(* CODESYS project heartbeat.2020.0113.1.project

Project tree, tasks and I/O mapping:
  Device : Changsha-Cyber-MI-linux, Changsha Cyber-MI Co., Ltd., version 3.5.10.40
    application Application
      libraries: Standard, * (System); SysFile, 3.5.9.0 (System); SysTypes2 Interfaces, * (System); SysShm, * (System); CAA Mathematics, * (CAA Technical Workgroup); SysTime, 3.5.9.0 (System); CAA Types Extern, 3.5.13.0 (CAA Technical Workgroup); TCP, 3.5.9.50 (3S - Smart Software Solutions GmbH); CAA Net Base Services, 3.5.14.0 (CAA Technical Workgroup); CAA DTUtil Extern, 3.5.12.0 (CAA Technical Workgroup); Util, * (System)
      task c_MainTask (cyclic, interval 10 ms, priority 20) calls prg_heartbeat, prg_data2file
      Enums/
        data type ERROR
        data type MQTT_STATE
        data type UDP_STATE_1
      data type UDP_STATE
      programs/
        program prg_heartbeat [ST]
      Function Blocks/
        function block FB_RETAIN [ST]: wr_all, SetDefault, chk_change, rd_all, is_default
        function block FB_MQTT_PUBLISH_CLIENT [ST]: m_fill_publish_buf, m_fill_connect_buf
        function block FB_DATA2FILE [ST]
      Functions/
        function Enable_120ohm_can0 [ST]
        function write_num_to_file [ST]
        function read_num_from_file [ST]
        function Enable_120ohm_can1 [ST]
        function Disable_120ohm_can0 [ST]
        function Disable_120ohm_can1 [ST]
        function Set_piv01 [ST]
        function Set_piv23 [ST]
        function set_ip [ST]
        function set_wifi_passwd [ST]
        function read_iccid [ST]
        function read_ip [ST]
        function read_sn [ST]
        function read_wifi_passwd [ST]
        function read_work_mins [ST]
        function read_location [ST]
      heartbeat/
        function fn_cyber_layer1 [ST]
        function fn_cyber_layer2 [ST]
        function fn_cyber_heartBeat [ST]
        function fn_sn_str_to_byte [ST]
        function Iccid_to_bytes [ST]
      GlobalConstants/
        global variables Constants
      program prg_data2file [ST]
    SoftMotion General Axis Pool
  libraries: VisuSymbols, 3.5.10.0 (System)
  5ce3da45-db07-42e7-a21c-a00fff4ed8f6|C:\Users\zhou\p01.bmp
  5ce3da45-db07-42e7-a21c-a00fff4ed8f6|C:\working\p01.bmp
  5ce3da45-db07-42e7-a21c-a00fff4ed8f6|C:\working\file.bmp
  text list GlobalTextList
*)

// Device/Application/UDP_STATE
TYPE UDP_STATE :
(
	INIT := 0, 	(* first State. Connections are set up *)
	SEND,		(* Send messages *)
	READ,		(* Receive messages *)
	ERROR		(* Prepare to reset connections *)
);
END_TYPE

// Device/Application/Enums/ERROR
{attribute 'qualified_only'}
//{attribute 'conditionalshow'}
//{attribute 'conditionalshow' := 'SomeText'}
//{attribute 'hide'}
TYPE ERROR : (NO_ERROR, TIME_OUT); END_TYPE

// Device/Application/Enums/MQTT_STATE
{attribute 'qualified_only'}
{attribute 'strict'}
TYPE MQTT_STATE :
(
	INIT := 0,
	CONN_SEND,
	CONN_RECV,
	READY,
	SEND,
	RECV,
	ERROR
);
END_TYPE

// Device/Application/Enums/UDP_STATE_1
TYPE UDP_STATE_1 :
(
	INIT := 0, 	(* first State. Connections are set up *)
	SEND,		(* Send messages *)
	READ,		(* Receive messages *)
	ERROR		(* Prepare to reset connections *)
);
END_TYPE

// Device/Application/GlobalConstants/Constants
{attribute 'qualified_only'}

VAR_GLOBAL CONSTANT
	RETAIN_NUM_MAX : INT := 256; 
END_VAR

// Device/Application/programs/prg_heartbeat
PROGRAM prg_heartbeat
VAR_OUTPUT
	lock_state :INT := 0;
	unlock_state :INT := 0;
	lock_unlock_level :INT := 0;
	delay_time :INT := 0;
END_VAR

VAR
	is_inited :BOOL := FALSE;
	eSTATE			: UDP_STATE; (* 状态转换变量 *)
	
	myIP		: NBS.IP_ADDR; (* MIC7001本身的IP地址 *)
	myPort		: UINT; (* MIC7001用于通信的端口 *)
	IPSend		: NBS.IP_ADDR; (* 对方的IP地址 *)
	PortSend	: UINT; (* 对方的端口 *)

	sToSend			: STRING; (* 待发送数据 *)
	sReceived		: STRING; (* 接收数据 *)
	
	UDPPeer			: NBS.UDP_Peer; (* FB UDP Peer *)
	UDPSend			: NBS.UDP_Send; (* FB UDP Send *)
	UDPReceive		: NBS.UDP_Receive; (* FB UDP Receive *)
	Peer			: CAA.HANDLE; (* Handle to the peer connection *)

	size :CAA.SIZE;	
	Writebuffer: 			ARRAY[1..200] OF BYTE;
	Readbuffer: 			ARRAY[0..1499] OF BYTE;
	ReadbufferStr: STRING;
	atcState :INT := 0;
	
	writeUdpState :INT := 0;
	readUdpState :INT := 0;
	
	i :INT;
	count :INT := 0;
	
	rtc_fb: RTC;
	dtu_set_dt_fb: dtu.SetDateAndTime;
	
	
	server_ip:STRING := '47.107.240.29';
	server_port:UINT := 34567;
	
	is_read :BOOL := FALSE;
	read_count :INT := 0;
	readFileState :INT := 0;
	ton_fb :TON;
	iccid_read_buffer :STRING;
	position :INT := -1;
	new_date:DT;
	iStat :UINT := 0;
	lac : STRING(4) := '0000';
	ci : STRING(4) := '0000';
	lenHearBeat:UINT;
	dataHearBeat:ARRAY[0..255] OF BYTE;
	ton_hb:ton; //heartbeat timer 
	bReturn:BOOL;
	lenLayer2:UINT;
	dataLayer2:ARRAY[0..255] OF BYTE;
	lenLayer1:UINT;
	lenRecvLayer1:UINT := 1500;
	dataLayer1:ARRAY[0..255] OF BYTE;
	bSN :ARRAY[0..6] OF BYTE;
	sub_str:STRING(8);
	num :UINT;
	lenHeartBeat: UINT;
	sn: STRING;
	work_time: DINT;
	dataIndex :UINT := 0;
	cntr_lac:UINT := 0;
	cntr_iccid:UINT := 0;
	cntr_recv:UINT := 0;
	dataLayern:ARRAY[1..255] OF BYTE;
	recv_size :CAA.SIZE;
	
	/// 辅助变量 
	xSend			: BOOL;
	sTmp1			: STRING;
	xEnable			: BOOL;	
	gprs_serial :CAA.HANDLE;
END_VAR

CASE iStat OF
0:
	xEnable:= TRUE;  //用于启动最下方的第70行的UDPPeer
	// 建立连接后马上转到发送状态
	IF UDPPeer.xActive THEN 
		eSTATE:= UDP_STATE.send;
	ELSIF UDPPeer.xError THEN
		eSTATE:= UDP_STATE.ERROR;
	END_IF
	
	IPSend.sAddr := server_ip;
	iStat := 2;
	
2:
	IF NOT read_iccid(ADR(iccid_read_buffer)) THEN
		iccid_read_buffer := 'iccid_null';		
	END_IF;
	iStat := 10;
	
10: //read sn
	IF NOT read_sn(ADR(sn)) THEN 
		sn := 'sn_null';
	END_IF
	
	iStat := 15;
	
15:
	read_location(ADR(lac), ADR(ci));
	iStat := 30;
30:
	work_time := read_work_mins();
	iStat := 100;
	
100:   //定时等待
	ton_fb(IN := TRUE, PT := T#10S);
	IF (ton_fb.Q) THEN
		ton_fb(IN := FALSE, PT := T#10S);
		iStat := 200;  //发送心跳
	ELSE
		iStat := 300; //发送实时数据	
	END_IF
	
200:
	bReturn := fn_cyber_heartBeat(	  //填充第三层：心跳帧
						lac_str := lac, 
						cid_str := ci, 
						ccid_str := iccid_read_buffer, 
						mins := work_time, 
						clientCode := 6,   //hengtian 95
						machineCode := 5,  //挖掘机
						pLenOut := ADR(lenHearBeat), 
						pDataOut := ADR(dataHearBeat)
	);
	
	IF NOT bReturn THEN
		RETURN;
	END_IF;

	dataIndex := dataIndex + 1;
	bReturn := fn_cyber_layer2( //填充第二层，数据层
						dataType := 1,
						paraId := 0,
						dataIndex := dataIndex,
						ver := 1,
						res1 := 0,
						LenIn := lenHearBeat,
						pDataIn := ADR(dataHearBeat),
						pLenOut := ADR(lenLayer2),
						pDataOut := ADR(dataLayer2)
	);
				
	IF NOT bReturn THEN
		RETURN;
	END_IF;

	bSN := fn_sn_str_to_byte(sn);
	bReturn := fn_cyber_layer1(    //填充第一层，设备层
						sn := ADR(bSN),
						ver := 1,
						lenIn := lenLayer2,
						pDataIn := ADR(dataLayer2),
						pLenOut := ADR(lenLayer1),
						pDataOut := ADR(dataLayer1)
	);
	
	IF NOT bReturn THEN
		RETURN;
	ELSE
		UDPSend(xExecute := FALSE);
		iStat := 500;
	END_IF;
	
300:  //sending realtime data  here
	//UDPSend(some realtime data as need);
	iStat := 100;
	
500:
	UDPSend(xExecute := TRUE, hPeer := Peer, ipAddr := IPSend, uiPort := server_port, szSize := lenLayer1, pDAta := ADR(dataLayer1));
	IF UDPSend.xDone THEN
		UDPSend(xExecute := FALSE);
		iStat := 600; 
	END_IF
	
	IF UDPSend.xError THEN  
		UDPSend(xExecute := FALSE);
		iStat := 30; 
	END_IF
	
	
600:
	UDPReceive(xEnable := TRUE, hPeer := Peer, szSize := SIZEOF(Readbuffer), pData := ADR(Readbuffer));
	IF UDPReceive.xDone THEN  //接收到数据
	 	recv_size := UDPReceive.szCount;
		UDPReceive(xEnable := FALSE);
		iStat := 30; //read mins and lca again
		IF recv_size = 25 THEN
			lock_state := BYTE_TO_INT(Readbuffer[20]);
			unlock_state := BYTE_TO_INT(Readbuffer[21]);
			lock_unlock_level := BYTE_TO_INT(Readbuffer[22]);
			delay_time := BYTE_TO_INT(Readbuffer[23]);
		END_IF
	ELSE
		cntr_recv := cntr_recv + 1;
		IF cntr_recv > 20 THEN
			cntr_recv := 0;
			iStat := 30;
		END_IF
	END_IF
	
	IF UDPReceive.xError THEN  //接收错误
		UDPReceive(xEnable := FALSE);
		recv_size := 0;
		iStat := 30; //read mins and lca again
	END_IF
END_CASE

//保持每个周期调用，维护与对方的连接关系本地端口的接收状态
UDPPeer(xEnable:= xEnable, hPeer=> Peer);
RETURN;

END_PROGRAM

// Device/Application/Functions/read_iccid
FUNCTION read_iccid : BOOL
VAR_INPUT
	iccid: POINTER TO STRING;
END_VAR

VAR
	hFile: RTS_IEC_HANDLE;
	udiOpenError: RTS_IEC_RESULT;
	udiReadError: RTS_IEC_RESULT;
	i :INT;
	iTemp: UDINT;
	udiPos: UDINT;
	str_size: __XWORD;
	udiByteRead: LWORD;

	len_of_line: INT;
	len_of_number :INT;
	magicNumber:REAL;
	check_sum:REAL:= 0;
	temp_num:REAL;
END_VAR

read_iccid := FALSE;

//检测文件是否存在
hFile := sysfileopen(szFile := '/userapp/iccid.txt', am := sysfile.AM_READ, pResult:= ADR(udiOpenError));
IF hFile = RTS_INVALID_HANDLE	THEN  //文件不存在
	RETURN;
END_IF
//文件存在，开始读取内容
udiPos := SysFileSetPos(hFile:=hFile, ulOffset := 0);
udiByteRead := sysfile.SysFileRead(hfile := hFile,pbyBuffer := iccid, ulSize := 32, pResult := ADR(udiReadError));
IF udiByteRead < 4 THEN  //读取失败
	sysfile.SysFileClose(hFile := hFile);
	RETURN;
END_IF

sysfile.SysFileClose(hFile := hFile);
read_iccid := TRUE;

END_FUNCTION

// Device/Application/Functions/read_sn
FUNCTION read_sn : BOOL
VAR_INPUT
	sn: POINTER TO STRING;
END_VAR

VAR
	hFile: RTS_IEC_HANDLE;
	udiOpenError: RTS_IEC_RESULT;
	udiReadError: RTS_IEC_RESULT;
	i :INT;
	iTemp: UDINT;
	udiPos: UDINT;
	str_size: __XWORD;
	udiByteRead: LWORD;

	len_of_line: INT;
	len_of_number :INT;
	magicNumber:REAL;
	check_sum:REAL:= 0;
	temp_num:REAL;
END_VAR

read_sn := FALSE;

//检测文件是否存在
hFile := sysfileopen(szFile := '/userapp/sn.txt', am := sysfile.AM_READ, pResult:= ADR(udiOpenError));
IF hFile = RTS_INVALID_HANDLE	THEN  //文件不存在
	RETURN;
END_IF
//文件存在，开始读取内容
udiPos := SysFileSetPos(hFile:=hFile, ulOffset := 0);
udiByteRead := sysfile.SysFileRead(hfile := hFile,pbyBuffer := sn, ulSize := 32, pResult := ADR(udiReadError));
IF udiByteRead < 4 THEN  //读取失败
	sysfile.SysFileClose(hFile := hFile);
	RETURN;
END_IF
sysfile.SysFileClose(hFile := hFile);
read_sn := TRUE;

END_FUNCTION

// Device/Application/Functions/read_location
FUNCTION read_location : BOOL
VAR_INPUT
	lac:POINTER TO STRING;
	ci:POINTER TO STRING;
END_VAR

VAR
	hFile: RTS_IEC_HANDLE;
	udiOpenError: RTS_IEC_RESULT;
	udiReadError: RTS_IEC_RESULT;
	i :INT;
	iTemp: UDINT;
	udiPos: UDINT;
	str_size: __XWORD;
	udiByteRead: LWORD;

	len_of_line: INT;
	len_of_number :INT;
	magicNumber:REAL;
	check_sum:REAL:= 0;
	temp_num:REAL;	
END_VAR

read_location := FALSE;
lac^ := '0000';
ci^ := '0000';

//检测文件是否存在
hFile := sysfileopen(szFile := '/userapp/laccid.txt', am := sysfile.AM_READ, pResult:= ADR(udiOpenError));
IF hFile = RTS_INVALID_HANDLE	THEN  //文件不存在
	RETURN;
END_IF

//文件存在，开始读取内容
udiPos := SysFileSetPos(hFile:=hFile, ulOffset := 0);
udiByteRead := sysfile.SysFileRead(hfile := hFile,pbyBuffer := lac, ulSize := 32, pResult := ADR(udiReadError));
IF udiByteRead < 4 THEN  //读取失败
	sysfile.SysFileClose(hFile := hFile);
	RETURN;
END_IF
sysfile.SysFileClose(hFile := hFile);

hFile := sysfileopen(szFile := '/userapp/cid.txt', am := sysfile.AM_READ, pResult:= ADR(udiOpenError));
IF hFile = RTS_INVALID_HANDLE	THEN  //文件不存在
	RETURN;
END_IF

//文件存在，开始读取内容
udiPos := SysFileSetPos(hFile:=hFile, ulOffset := 0);
udiByteRead := sysfile.SysFileRead(hfile := hFile,pbyBuffer := ci, ulSize := 32, pResult := ADR(udiReadError));
IF udiByteRead < 4 THEN  //读取失败
	sysfile.SysFileClose(hFile := hFile);
	RETURN;
END_IF
sysfile.SysFileClose(hFile := hFile);

read_location := TRUE;

END_FUNCTION

// Device/Application/Functions/read_work_mins
FUNCTION read_work_mins : DINT;
VAR_INPUT
END_VAR

VAR
	time_file_name :STRING := '/userapp/r_mins.txt';
	hFile: RTS_IEC_HANDLE;
	udiOpenError: RTS_IEC_RESULT;
	udiReadError: RTS_IEC_RESULT;

	udiPos: UDINT;
	str_size: __XWORD;
	udiByteRead: LWORD;
	read_buf:STRING;

END_VAR

read_work_mins := 0;

//检测文件是否存在
hFile := sysfileopen(szFile := time_file_name, am := sysfile.AM_READ, pResult:= ADR(udiOpenError));
IF hFile = RTS_INVALID_HANDLE	THEN  //文件不存在
	RETURN;
END_IF

//文件存在，开始读取内容
udiPos := SysFileSetPos(hFile:=hFile, ulOffset := 0);
udiByteRead := sysfile.SysFileRead(hfile := hFile,pbyBuffer := ADR(read_buf), ulSize := 32, pResult := ADR(udiReadError));
sysfile.SysFileClose(hFile := hFile);

read_work_mins := ANY_TO_DINT(read_buf);

END_FUNCTION

// Device/Application/heartbeat/fn_cyber_heartBeat
FUNCTION fn_cyber_heartBeat : bool
VAR_INPUT
	lac_str:STRING(4);
	cid_str:STRING(4);
	ccid_str:STRING(21);
	mins:UDINT;
	clientCode:UINT;
	machineCode:UINT;
	pLenOut:POINTER TO UINT;
	pDataOut:POINTER TO BYTE;
END_VAR
VAR
	index: UINT;
	data_uint: UINT;
	data_byte_array:ARRAY[0..9] OF BYTE;
	i: INT;
END_VAR

fn_cyber_heartBeat := FALSE;

index := 0;
data_uint := STRING_TO_UINT(concat('16#',lac_str));
pDataOut[index] := ANY_TO_BYTE(data_uint/256);
index := index + 1;

pDataOut[index] := ANY_TO_BYTE(data_uint MOD 256);
index := index + 1;

data_uint := STRING_TO_UINT(concat('16#',cid_str));
pDataOut[index] := ANY_TO_BYTE(data_uint/256);
index := index + 1;

pDataOut[index] := ANY_TO_BYTE(data_uint MOD 256);
index := index + 1;

data_byte_array := Iccid_to_bytes(ccid_str);
FOR i := 0 TO 9 DO
	pDataOut[index] := data_byte_array[i];
	index := index + 1;
END_FOR

pDataOut[index] := ANY_TO_BYTE(mins/256/256/256);
index := index + 1;

pDataOut[index] := ANY_TO_BYTE(mins/256/256);
index := index + 1;

pDataOut[index] := ANY_TO_BYTE(mins/256);
index := index + 1;

pDataOut[index] := ANY_TO_BYTE(mins);
index := index + 1;

pDataOut[index] := ANY_TO_BYTE(clientCode/256);
index := index + 1;

pDataOut[index] := ANY_TO_BYTE(clientCode);
index := index + 1;

pDataOut[index] := ANY_TO_BYTE(machineCode/256);
index := index + 1;

pDataOut[index] := ANY_TO_BYTE(machineCode);
index := index + 1;

pLenOut^ := index;

fn_cyber_heartBeat := TRUE;

END_FUNCTION

// Device/Application/heartbeat/Iccid_to_bytes
FUNCTION Iccid_to_bytes : ARRAY[0..9] OF BYTE
VAR_INPUT
	iccd :STRING;
END_VAR
VAR
	iccid_code :ARRAY[0..9] OF BYTE;
	
	byteHigh :BYTE := 0;
	byteLow :BYTE := 0;
	dstLen :INT := 0;
	
	srcIndex :INT := 0;
	bytesIndex :INT := 0;
	sub_str:STRING(32);
END_VAR

dstLen := len(iccd) / 2;

sub_str := iccd;
FOR bytesIndex := 0 TO dstLen - 1 DO
	iccid_code[bytesIndex] := BYTE_TO_BCD(STRING_TO_BYTE(left(sub_str,2)));	
	sub_str := delete(sub_str,2,1);
END_FOR

Iccid_to_bytes := iccid_code;

END_FUNCTION

// Device/Application/heartbeat/fn_cyber_layer2
FUNCTION fn_cyber_layer2 : bool
VAR_INPUT
	dataType : BYTE := 0;
	paraId :BYTE := 0;
	dataIndex : UINT := 0;
	ver :BYTE := 1;
	res1 :BYTE := 0;
	LenIn :UINT := 0;
	pDataIn :POINTER TO BYTE;
	pLenOut :POINTER TO UINT;
	pDataOut :POINTER TO BYTE;
END_VAR
VAR
	i:UINT:= 0;
	index:UINT := 0;
END_VAR

fn_cyber_layer2 := FALSE;

index := 0;
pDataOut[index] := dataType;
index := index + 1;

pDataOut[index] := paraId;
index := index + 1;

pDataOut[index] := ANY_TO_BYTE(dataIndex/256);
index := index + 1;

pDataOut[index] := ANY_TO_BYTE(dataIndex MOD 256);
index := index + 1;

pDataOut[index] := ver;
index := index + 1;

pDataOut[index] := res1;
index := index + 1;

pDataOut[index] := ANY_TO_BYTE(LenIn/256);
index := index + 1;

pDataOut[index] := ANY_TO_BYTE(LenIn MOD 256);
index := index + 1;

FOR i := 0 TO LenIn-1 DO
	pDataOut[index] := pDataIn[i];
	index := index + 1;
END_FOR

pLenOut^ := index;

fn_cyber_layer2 := TRUE;
RETURN;

END_FUNCTION

// Device/Application/heartbeat/fn_sn_str_to_byte
FUNCTION fn_sn_str_to_byte : ARRAY[0..6] OF BYTE
VAR_INPUT
	sn:STRING(16);
END_VAR
VAR
	i: INT;
	bSN: ARRAY[0..6] OF BYTE;
	sub_str: STRING(255);
	num: UINT;
	bcd: UINT;
END_VAR

// 1.2 12
sub_str := mid(sn, 2, 4);
bcd := STRING_TO_UINT(sub_str);
bcd := (bcd / 10) *16 + (bcd MOD 10);
bSN[0] := UINT_TO_BYTE(bcd);

// 1.3 34
sub_str := mid(sn, 2, 6);
bcd := STRING_TO_UINT(sub_str);
bcd := (bcd / 10) *16 + (bcd MOD 10);
bSN[1] := UINT_TO_BYTE(bcd);

// 1.4 56
sub_str := mid(sn, 2, 8);
bcd := STRING_TO_UINT(sub_str);
bcd := (bcd / 10) *16 + (bcd MOD 10);
bSN[2] := UINT_TO_BYTE(bcd);

// 1.5 78
sub_str := mid(sn, 2, 10);
bcd := STRING_TO_UINT(sub_str);
bcd := (bcd / 10) *16 + (bcd MOD 10);
bSN[3] := UINT_TO_BYTE(bcd);

// 1.6 1234
sub_str := mid(sn, 2, 12);
bcd := STRING_TO_UINT(sub_str);
bcd := (bcd / 10) *16 + (bcd MOD 10);
bSN[4] := UINT_TO_BYTE(bcd);

sub_str := mid(sn, 2, 14);
bcd := STRING_TO_UINT(sub_str);
bcd := (bcd / 10) *16 + (bcd MOD 10);
bSN[5] := UINT_TO_BYTE(bcd);

fn_sn_str_to_byte := bSN;

END_FUNCTION

// Device/Application/heartbeat/fn_cyber_layer1
FUNCTION fn_cyber_layer1 : bool
VAR_INPUT
	sn:POINTER TO BYTE;
	ver:BYTE := 0;
	lenIn:UINT := 0;
	pDataIn:POINTER TO BYTE;
	pLenOut:POINTER TO UINT ;
	pDataOut: POINTER TO BYTE;
END_VAR
VAR
	i:UINT;
	index:UINT;
	checksum:UINT;
END_VAR

fn_cyber_layer1 := FALSE;

index := 0;
checksum := 0;
FOR i := 0 TO 8 DO
	pDataOut[index] := sn[i];
	index := index+1;
	checksum := checksum + sn[i];
END_FOR

pDataOut[index] := ver;
index := index+1;
checksum := checksum + ver;

pDataOut[index] := ANY_TO_BYTE(lenIn/256);
index := index+1;
checksum := checksum + ANY_TO_BYTE(lenIn/256);

pDataOut[index] := ANY_TO_BYTE(lenIn MOD 256);
index := index+1;
checksum := checksum + ANY_TO_BYTE(lenIn MOD 256);

FOR i := 0 TO lenIn-1 DO
	pDataOut[index] := pDataIn[i];
	index := index+1;	
	checksum := checksum + pDataIn[i];
END_FOR

pDataOut[index] := ANY_TO_BYTE(checksum/256);
index := index+1;

pDataOut[index] := ANY_TO_BYTE(checksum MOD 256);
index := index+1;

pLenOut^ := index;

fn_cyber_layer1 := TRUE;

END_FUNCTION

// Device/Application/prg_data2file
PROGRAM prg_data2file
VAR
	data:ARRAY[0..255] OF REAL;
	data2file :FB_DATA2FILE;
	
	init:BOOL:= FALSE;
	hFile: RTS_IEC_HANDLE := RTS_INVALID_HANDLE;
	udiOpenError: RTS_IEC_RESULT;
	udiWriteError: RTS_IEC_RESULT;
	str:STRING := 'asdf';
	sizewrite:dword;
END_VAR

data2file(data := data, length := 28, interval := T#300MS, filename := '/userdata/test_data_001.csv', maxsize_m := 15);



IF NOT init THEN
	hFile := sysfileopen(szFile := '/userapp/cmux', am := sysfile.AM_WRITE, pResult := ADR(udiOpenError));
	sizewrite := sysfile.SysFileWrite(hFile := hFile,pbyBuffer := ADR(str),ulSize := 4, pResult := ADR(udiWriteError));
	sysfile.SysFileClose(hFile);
	init := TRUE;
END_IF

END_PROGRAM

// Device/Application/Function Blocks/FB_DATA2FILE
FUNCTION_BLOCK FB_DATA2FILE
VAR_INPUT
	xEnable:BOOL := FALSE;
	data:ARRAY[0..255] OF REAL;
    length:DINT;
    interval:TIME := T#100MS; 
	filename:STRING := '/userdata/data_01.csv';
	maxsize_m:DINT := 1;
END_VAR

VAR_OUTPUT
	xFull:BOOL := FALSE;
	xBusy:BOOL := FALSE;
	xError:BOOL := FALSE;
	udiFilesize:UDINT := 0;
END_VAR

VAR
	iStat :UINT := 0;
	udiDeleteError: RTS_IEC_RESULT;
	udiOpenError: RTS_IEC_RESULT;
	udiWriteError: RTS_IEC_RESULT;
	udiSizeError: RTS_IEC_RESULT;	
	hFile: RTS_IEC_HANDLE := RTS_INVALID_HANDLE;
	tmr_wr:ton();
	filesize: __XWORD;
	i :DWORD;
	iTemp: UDINT;
	udiPos: UDINT;	
	str: STRING(256);
	str_size: __XWORD;
	udiByteWrite: LWORD;
END_VAR


CASE iStat OF
0:
	xFull := FALSE;
	xBusy := FALSE;
	xError := FALSE;
	udiFilesize := 0;
	IF NOT xEnable THEN
		RETURN;
	ELSE
		iStat := 10;
	END_IF

10:
	hFile := sysfileopen(szFile := filename, am := sysfile.AM_APPEND_PLUS, pResult := ADR(udiOpenError));
 	IF hFile = RTS_INVALID_HANDLE	THEN  //打开文件失败
		xError := TRUE;
		RETURN;
	ELSE
		filesize := sysfilegetsize(filename, ADR(udiSizeError));
		IF filesize/1000000 > maxsize_m THEN
			iStat := 30;
		END_IF
		iStat := 20;
	END_IF	
	
20:
	tmr_wr(in := NOT tmr_wr.Q, pt := interval);
	IF tmr_wr.Q THEN
		filesize := sysfilegetsize(filename, ADR(udiSizeError));
		udiPos := SysFileSetPos(hFile:=hFile, ulOffset:=filesize);	
		udiFilesize := filesize;
		
		str:= '';
		FOR i := 0 TO length-1 DO
			str := concat(str, REAL_TO_STRING(data[i]));
			str := concat(str, ',');
			str_size := ANY_TO_DWORD(len(str));
			udiFilesize := udiFilesize + str_size;
			IF str_size > 200 THEN
				udiByteWrite := sysfile.SysFileWrite(hFile := hFile,pbyBuffer := ADR(str),ulSize := str_size, pResult := ADR(udiWriteError));
				IF udiByteWrite = str_size THEN
					str := '';
				END_IF
			END_IF
		END_FOR
		
		str := concat(str, '$N');	
		udiFilesize := udiFilesize + 1;	
		str_size := ANY_TO_DWORD(len(str));
		udiByteWrite := sysfile.SysFileWrite(hFile := hFile,pbyBuffer := ADR(str),ulSize := str_size, pResult := ADR(udiWriteError));
		IF udiFilesize/1000000 > maxsize_m THEN
			iStat := 30;
		END_IF
	END_IF 

30:
	xFull := TRUE;
	xError := TRUE;
	sysfileclose(hFile := hFile);
	iSTat := 40;
40:
	
END_CASE

IF NOT xEnable THEN
	sysfileclose(hFile := hFile);
	iStat := 0;
	RETURN;
END_IF

END_FUNCTION_BLOCK

// Device/Application/Function Blocks/FB_RETAIN
FUNCTION_BLOCK FB_RETAIN
VAR_INPUT
	set_default:BOOL := FALSE;
	default_val:ARRAY[0..Constants.RETAIN_NUM_MAX] OF DINT;
	filename:STRING[64];
END_VAR
VAR_IN_OUT
	value:ARRAY[0..Constants.RETAIN_NUM_MAX] OF DINT;
END_VAR
VAR_OUTPUT
	ok:BOOL := FALSE;
	err:BOOL := FALSE;
	default: BOOL := FALSE;
	err_code:DINT := 0;
END_VAR
VAR
	hFile: RTS_IEC_HANDLE := 0;
	sync:BOOL := FALSE;  
	stat:UINT:= 0;
	old_val:ARRAY[0..Constants.RETAIN_NUM_MAX] OF DINT;
	para_number:DINT := Constants.RETAIN_NUM_MAX;
	i: DINT;
	ret_val :BOOL := FALSE;
END_VAR

IF NOT ok THEN
	ret_val := rd_all();
	IF ret_val THEN
		ok := TRUE;
		err := FALSE;
		default := is_default();
	ELSE
		ret_val := SetDefault();
		IF ret_val THEN
			default := TRUE;
			ok := TRUE;
			err := FALSE;
		ELSE
			ok := FALSE;
			err := TRUE;
			default := FALSE;
			err_code := -1;
			RETURN;
		END_IF
	END_IF
END_IF

IF set_default THEN
	SetDefault();
	set_default := FALSE;
	default := TRUE;
	ok := TRUE;
	err := FALSE;
END_IF

IF chk_change() THEN
	wr_all();
END_IF

METHOD wr_all : bool
VAR_INPUT
END_VAR

VAR
	iNumber:INT;
	udiByteWrite:LWORD;
	udiPos:UDINT;
	udiOpenError: RTS_IEC_RESULT;
	udiWriteError: RTS_IEC_RESULT;
	str_size:DWORD;
	str: STRING(255);
	check_sum: DINT;
	i:DINT;
	
END_VAR
wr_all := FALSE;
hFile := sysfileopen(szFile := filename, am := sysfile.AM_WRITE, pResult := ADR(udiOpenError));
IF hFile = RTS_INVALID_HANDLE THEN
	RETURN;
END_IF

udiPos := SysFileSetPos(hFile:=hFile, ulOffset := 0);

check_sum := 0;
str:= ANY_TO_STRING('');
FOR i := 0 TO para_number DO
	IF i = para_number THEN  //the last val, check_sum
		value[i] := check_sum;
	ELSE
		check_sum := check_sum + value[i];
	END_IF
	str := concat(str, ANY_TO_STRING(value[i]));
	str := concat(str, ANY_TO_STRING('$N'));
	str_size := ANY_TO_DWORD(len(str));
	IF str_size > 200 THEN
		udiByteWrite := sysfile.SysFileWrite(hFile := hFile,pbyBuffer := ADR(str),ulSize := str_size, pResult := ADR(udiWriteError));
		IF udiByteWrite = str_size THEN
			str := '';
		END_IF
	END_IF	
END_FOR
udiByteWrite := sysfile.SysFileWrite(hFile := hFile,pbyBuffer := ADR(str),ulSize := str_size, pResult := ADR(udiWriteError));
	
IF udiByteWrite <> str_size THEN
	sysfile.SysFileClose(hFile);
	RETURN;
END_IF
sysfile.SysFileClose(hFile);
	
FOR i := 1 TO para_number DO
	old_val[i] := value[i];
END_FOR

hFile := 0;

wr_all := TRUE;
END_METHOD

METHOD SetDefault : bool
VAR_INPUT
END_VAR

VAR
	
END_VAR
SetDefault := FALSE;

FOR i := 0 TO para_number DO
	old_val[i] := default_val[i];
	value[i] := default_val[i];
END_FOR

SetDefault := wr_all();

RETURN;
END_METHOD

METHOD chk_change : bool
VAR_INPUT
END_VAR

VAR

END_VAR
chk_change := TRUE;

FOR i := 0 TO para_number DO
	IF value[i] <> old_val[i] THEN
		RETURN;
	END_IF
END_FOR

chk_change := FALSE;
END_METHOD

METHOD rd_all : bool
VAR_INPUT
END_VAR

VAR
	iNumber:INT;
	udiByteRead:LWORD;
	udiPos:UDINT;
	udiOpenError: RTS_IEC_RESULT;
	udiReadError: RTS_IEC_RESULT;
	str: STRING(255);
	ulOffset:DWORD;
	batch: BOOL;
	check_sum: DINT;
END_VAR
rd_all := FALSE;

hFile := sysfileopen(szFile := filename, am := sysfile.AM_READ, pResult:= ADR(udiOpenError));
IF hFile = RTS_INVALID_HANDLE THEN
	RETURN;
END_IF

ulOffset := 0;
batch := TRUE;

check_sum := 0;
FOR i := 0 TO para_number DO
	IF udiByteRead < 50 AND batch THEN
		udiPos := SysFileSetPos(hFile:=hFile, ulOffset := ulOffset);
		udiByteRead := sysfile.SysFileRead(hfile := hFile,pbyBuffer := ADR(str), ulSize := 255 , pResult := ADR(udiReadError));
		IF udiByteRead < 255 THEN
			batch := FALSE;
		END_IF
	END_IF
	IF udiByteRead < 1 THEN  //读取失败
		sysfile.SysFileClose(hFile := hFile);
		RETURN;
	END_IF

	iNumber := find(str, '$N');
	IF iNumber < 2 THEN
		sysfile.SysFileClose(hFile := hFile);
		RETURN;
	END_IF
	
	value[i] := STRING_TO_DINT(left(str,iNumber-1));
	str := delete(str, iNumber,1);
	old_val[i] := value[i];
	
	udiByteRead := udiByteRead - ANY_TO_LWORD(iNumber);
	ulOffset := ulOffset + ANY_TO_DWORD(iNumber);

	IF i = para_number THEN
		IF check_sum <> value[i] THEN
			sysfile.SysFileClose(hFile := hFile);
			RETURN;  //error
		END_IF
	ELSE
		check_sum := check_sum + value[i];
	END_IF
END_FOR

sysfile.SysFileClose(hFile := hFile);
rd_all := TRUE;
END_METHOD

METHOD is_default : bool
VAR_INPUT
END_VAR
is_default := FALSE;

FOR i := 0 TO para_number DO
	IF value[i] <> default_val[i] THEN
		RETURN;
	END_IF
END_FOR

is_default := TRUE;
END_METHOD

END_FUNCTION_BLOCK

// Device/Application/Function Blocks/FB_MQTT_PUBLISH_CLIENT
FUNCTION_BLOCK FB_MQTT_PUBLISH_CLIENT
VAR_INPUT
	s_svr_ip : STRING(32) := '47.107.240.29';
	ui_svr_port: UINT := 1883;
	s_client_id : STRING(255) := 'mic7001_test_id';
	s_topic:STRING(255) := 'mic7001_test_topic';
	s_payload:STRING(255):= 'mic7001_test_payload';
	ui_keep_alive:UINT := 60;
	xExecute:BOOL := FALSE;
END_VAR
VAR_OUTPUT
	stat:MQTT_STATE := MQTT_STATE.INIT;
	xError:BOOL := FALSE;
	xBusy:BOOL := FALSE;
	xDone:BOOL := FALSE;
END_VAR
VAR
	e_state : MQTT_STATE := MQTT_STATE.INIT;
	server_ip : NBS.IP_ADDR;
	server_port : UINT;
	udi_time_out : UDINT;
	mqtt_client : NBS.TCP_Client;
	mqtt_connection : CAA.HANDLE;
	mqtt_send : NBS.TCP_Write;
	mqtt_recv : NBS.TCP_Read;
	s_send_buf : ARRAY[0..255] OF BYTE;
	s_recv_buf : ARRAY[0..255] OF BYTE;
	buf_size :UINT := 0;
	i : INT;
	send_cmd :R_TRIG;
	conn_recv_cntr :UINT := 0;
	cntr :UINT := 0;
END_VAR

CASE e_state OF
	MQTT_STATE.INIT:
		xDone := FALSE;
		xError := FALSE;
		xBusy := FALSE;
		
		server_ip.sAddr := s_svr_ip;
		server_port := ui_svr_port;
	
		IF mqtt_client.xActive = TRUE THEN
			buf_size := m_fill_connect_buf();
			IF buf_size > 0 THEN
				mqtt_send.szSize := buf_size;
				mqtt_send(xExecute := FALSE);
				mqtt_send.xExecute := TRUE;
				mqtt_recv(xEnable := FALSE);
				mqtt_recv.xEnable := TRUE;
				e_state := MQTT_STATE.CONN_SEND;
				cntr := 0;
			ELSE
				e_state := MQTT_STATE.error;	
			END_IF
		ELSIF mqtt_client.xError = TRUE THEN
			e_state := MQTT_STATE.ERROR;
		ELSE
			cntr := cntr + 1;
			IF cntr > 100 THEN
				cntr := 0;
				e_state := MQTT_STATE.ERROR;
			END_IF
		END_IF
		
	MQTT_STATE.CONN_SEND:
		IF mqtt_send.xDone THEN
			e_state := MQTT_STATE.CONN_RECV;
			cntr := 0;
		ELSIF cntr > 100 THEN
			e_state := MQTT_STATE.ERROR;
		END_IF	
		cntr := cntr + 1;
	
	MQTT_STATE.CONN_RECV:
		IF mqtt_recv.xReady = TRUE AND s_recv_buf[0]=16#20 THEN
			e_state := MQTT_STATE.READY;
		ELSIF cntr > 100 THEN
			e_state := MQTT_STATE.ERROR;
		END_IF
		cntr := cntr + 1;
	
	MQTT_STATE.READY:
		send_cmd(clk := xExecute);
		IF send_cmd.Q THEN
			buf_size := m_fill_publish_buf();
			IF buf_size > 0 THEN
				mqtt_send.szSize := buf_size;
				mqtt_send(xexecute := FALSE);
				mqtt_send.xExecute := TRUE;
				e_state := MQTT_STATE.SEND;	
				cntr := 0;		
			ELSE
				e_state := MQTT_STATE.error;			
			END_IF
		END_IF
		
	MQTT_STATE.SEND:
		IF mqtt_send.xdone THEN
			e_state := MQTT_STATE.READY;
		ELSIF cntr > 100 THEN
			e_state := MQTT_STATE.ERROR;
		END_IF
		cntr := cntr + 1;
		(*
	MQTT_STATE.RECV:
		*)
	MQTT_STATE.ERROR:
		IF NOT xExecute THEN
			mqtt_client(xEnable := FALSE);
			mqtt_send(xExecute := FALSE);
			e_state := MQTT_STATE.INIT;
			xError := FALSE;
		END_IF
		xError := TRUE;
END_CASE


mqtt_client(xEnable := TRUE, ipAddr := server_ip, uiPort := server_port, udiTimeOut := 0, hConnection => mqtt_connection);
IF mqtt_connection > 0 THEN
	mqtt_send(udiTimeOut := udi_time_out, hConnection := mqtt_connection, pData := ADR(s_send_buf));
	mqtt_recv(hConnection := mqtt_connection, szSize := 64, pData := ADR(s_recv_buf));
END_IF
stat := e_state;

METHOD m_fill_publish_buf : UINT
VAR_INPUT
END_VAR

VAR
	i : UINT;
	ui_client_id_len : UINT;
	ui_topic_len :UINT;
	ui_payload_len:UINT;
	ui_mqtt_msg_len:UINT;
END_VAR
ui_topic_len := INT_TO_UINT(LEN(s_topic));
ui_payload_len := INT_TO_UINT(LEN(s_payload));
ui_mqtt_msg_len := ui_topic_len + ui_payload_len + 2;

// Header Flag. Publish command.
s_send_buf[0] := 16#30;
IF ui_mqtt_msg_len < 128 THEN
	// Msg Len.
	s_send_buf[1] := UINT_TO_BYTE(ui_mqtt_msg_len);
	// Topic Length.
	s_send_buf[2] := UINT_TO_BYTE(ui_topic_len / 256);
	s_send_buf[3] := UINT_TO_BYTE(ui_topic_len MOD 256);
	// Topic.
	FOR i:=0 TO ui_topic_len-1 DO
		s_send_buf[i + 4] := s_topic[i];
	END_FOR
	// Payload.
	FOR i:=0 TO ui_payload_len-1 DO
		s_send_buf[i + 4 + ui_topic_len] := s_payload[i];
	END_FOR
	ui_mqtt_msg_len := ui_mqtt_msg_len + 2;
	m_fill_publish_buf := ui_mqtt_msg_len;
ELSIF  ui_mqtt_msg_len < 16384 THEN
	// Msg Len.
	s_send_buf[1] := UINT_TO_BYTE(16#80 + ui_mqtt_msg_len - (ui_mqtt_msg_len / 128) * 128);
	s_send_buf[2] := UINT_TO_BYTE(ui_mqtt_msg_len / 128);
	// Topic Length.
	s_send_buf[3] := UINT_TO_BYTE(ui_topic_len / 256);
	s_send_buf[4] := UINT_TO_BYTE(ui_topic_len MOD 256);
	// Topic.
	FOR i:=0 TO LEN(s_topic)-1 BY 1 DO
		s_send_buf[i + 5] := s_topic[i];
	END_FOR
	// Payload.
	FOR i:=0 TO LEN(s_payload)-1 BY 1 DO
		s_send_buf[i + 5 + LEN(s_topic)] := s_payload[i];
	END_FOR
	ui_mqtt_msg_len := ui_mqtt_msg_len + 3;
	m_fill_publish_buf := ui_mqtt_msg_len;
ELSE
	m_fill_publish_buf := 0;
END_IF
END_METHOD

METHOD m_fill_connect_buf : UINT
VAR_INPUT
END_VAR

VAR
	ui_client_id_len : UINT;	
END_VAR
ui_client_id_len := INT_TO_UINT(LEN(s_client_id));
// Header Flag. Connect command.
s_send_buf[0] := 16#10;
// Msg Len.
s_send_buf[1] := UINT_TO_BYTE(12 + ui_client_id_len);
// Protocal Name Length.
s_send_buf[2] := 16#00;
s_send_buf[3] := 16#04;
// Protocal Name.
s_send_buf[4] := 16#4D;
s_send_buf[5] := 16#51;
s_send_buf[6] := 16#54;
s_send_buf[7] := 16#54;
// Version.
s_send_buf[8] := 16#04;
// Connect Flags.
s_send_buf[9] := 16#02;
// Keep Alive.
s_send_buf[10] := UINT_TO_BYTE(ui_keep_alive / 256);
s_send_buf[11] := UINT_TO_BYTE(ui_keep_alive MOD 256);
// Client ID Length.
s_send_buf[12] := UINT_TO_BYTE(ui_client_id_len / 256);
s_send_buf[13] := UINT_TO_BYTE(ui_client_id_len MOD 256);
// Client ID.
FOR i:=0 TO ui_client_id_len-1 DO
	s_send_buf[i+14] := s_client_id[i];
END_FOR

m_fill_connect_buf := ui_client_id_len+14;
END_METHOD

END_FUNCTION_BLOCK

// Device/Application/Functions/Enable_120ohm_can0
FUNCTION Enable_120ohm_can0 : BOOL
VAR_INPUT
END_VAR
VAR
	filename:STRING(32) := '/userapp/can0_r_en.txt';
END_VAR

Enable_120ohm_can0 := FALSE;

IF read_num_from_file(filename := filename) < 1 THEN
	Enable_120ohm_can0 := write_num_to_file(filename := filename, num := 1);
END_IF

RETURN;

END_FUNCTION

// Device/Application/Functions/read_num_from_file
FUNCTION read_num_from_file : dint
VAR_INPUT
	filename:STRING(32);
END_VAR
VAR
	hFile: RTS_IEC_HANDLE := 0;
	udiOpenError: RTS_IEC_RESULT;
	udiReadError: RTS_IEC_RESULT;
	rdbuf:STRING(32);	
END_VAR

read_num_from_file := -1;

hFile := sysfileopen(szFile := filename, am := sysfile.AM_READ, pResult:= ADR(udiOpenError));
IF hFile = RTS_INVALID_HANDLE THEN
	RETURN;
END_IF

SysFileSetPos(hFile:=hFile, ulOffset := 0);
sysfileread(hFile := hFile, pbyBuffer := ADR(rdbuf), ulSize := SIZEOF(rdbuf), pResult := ADR(udiReadError));
sysfileClose(hFile);

read_num_from_file := ANY_TO_DINT(rdbuf);
RETURN;

END_FUNCTION

// Device/Application/Functions/write_num_to_file
FUNCTION write_num_to_file : BOOL
VAR_INPUT
	filename:STRING(32);
	num:DINT;
END_VAR
VAR
	hFile: RTS_IEC_HANDLE := 0;
	udiOpenError: RTS_IEC_RESULT;
	udiWriteError: RTS_IEC_RESULT;
	wrbuf:STRING(32);
END_VAR

write_num_to_file := FALSE;

hFile := sysfileopen(szFile := filename, am := sysfile.AM_WRITE, pResult:= ADR(udiOpenError));
IF hFile = RTS_INVALID_HANDLE THEN
	RETURN;
END_IF

wrbuf := ANY_TO_STRING(num);
wrbuf := concat(wrbuf, '$n');
SysFileSetPos(hFile:=hFile, ulOffset := 0);
sysfilewrite(hFile := hFile, pbyBuffer := ADR(wrbuf), ulSize := len(wrbuf), pResult := ADR(udiWriteError));
sysfileClose(hFile);

write_num_to_file := TRUE;

RETURN;

END_FUNCTION

// Device/Application/Functions/Enable_120ohm_can1
FUNCTION Enable_120ohm_can1 : BOOL
VAR_INPUT
END_VAR
VAR
	filename:STRING(32) := '/userapp/can1_r_en.txt';
END_VAR

Enable_120ohm_can1 := FALSE;

IF read_num_from_file(filename := filename) < 1 THEN
	Enable_120ohm_can1 := write_num_to_file(filename := filename, num := 1);
END_IF

RETURN;

END_FUNCTION

// Device/Application/Functions/Disable_120ohm_can0
FUNCTION Disable_120ohm_can0 : BOOL
VAR_INPUT
END_VAR
VAR
	filename:STRING(32) := '/userapp/can0_r_en.txt';
	num :DINT;
END_VAR

Disable_120ohm_can0 := FALSE;

num := read_num_from_file(filename := filename);
IF  NOT (num = 0)  THEN
	Disable_120ohm_can0 := write_num_to_file(filename := filename, num := 0);
END_IF

RETURN;

END_FUNCTION

// Device/Application/Functions/Disable_120ohm_can1
FUNCTION Disable_120ohm_can1 : BOOL
VAR_INPUT
END_VAR
VAR
	filename:STRING(32) := '/userapp/can1_r_en.txt';
	num :DINT;
END_VAR

Disable_120ohm_can1 := FALSE;

num := read_num_from_file(filename := filename);
IF  NOT (num = 0)  THEN
	Disable_120ohm_can1 := write_num_to_file(filename := filename, num := 0);
END_IF

RETURN;

END_FUNCTION

// Device/Application/Functions/Set_piv01
FUNCTION Set_piv01 : BOOL
VAR_INPUT
	piv_mv:DINT := 10000;  // default: 10V
END_VAR
VAR
	filename:STRING(32) := '/userapp/piv01_mv.txt';
END_VAR

Set_piv01 := FALSE;

IF read_num_from_file(filename := filename) <> piv_mv THEN
	Set_piv01 := write_num_to_file(filename := filename, num := piv_mv);
END_IF

RETURN;

END_FUNCTION

// Device/Application/Functions/Set_piv23
FUNCTION Set_piv23 : BOOL
VAR_INPUT
	piv_mv:DINT := 10000;  // default: 10V
END_VAR
VAR
	filename:STRING(32) := '/userapp/piv23_mv.txt';
END_VAR

Set_piv23 := FALSE;

IF read_num_from_file(filename := filename) <> piv_mv THEN
	Set_piv23 := write_num_to_file(filename := filename, num := piv_mv);
END_IF

RETURN;

END_FUNCTION

// Device/Application/Functions/set_ip
FUNCTION set_ip : BOOL
VAR_INPUT
	ip: POINTER TO STRING;
END_VAR
VAR
	hFile: RTS_IEC_HANDLE;
	udiOpenError: RTS_IEC_RESULT;
	udiReadError: RTS_IEC_RESULT;
	udiWriteError: RTS_IEC_RESULT;
	i :INT;
	iTemp: UDINT;
	udiPos: UDINT;
	str_size: __XWORD;
	udiByteRead: UDINT;
	length:DINT;
	
	len_of_line: INT;
	len_of_number :INT;
	magicNumber:REAL;
	check_sum:REAL:= 0;
	temp_num:REAL;
	udiByteWrite: LWORD;
END_VAR


set_ip := FALSE;

hFile := sysfileopen(szFile := '/userapp/ipaddr.txt', am := sysfile.AM_WRITE, pResult := ADR(udiOpenError));
IF hFile = RTS_INVALID_HANDLE THEN //创建文件失败
	RETURN;
END_IF

length := LEN(ip);
udiPos := SysFileSetPos(hFile:=hFile, ulOffset:=0);	
udiByteWrite := sysfile.SysFileWrite(hFile := hFile,pbyBuffer := ip,ulSize := length, pResult := ADR(udiWriteError));
IF udiByteWrite = 0 THEN
	sysfile.SysFileClose(hFile := hFile);
	RETURN;
END_IF
sysfile.SysFileClose(hFile := hFile);
set_ip := TRUE;
RETURN;

END_FUNCTION

// Device/Application/Functions/set_wifi_passwd
FUNCTION set_wifi_passwd : BOOL
VAR_INPUT
	passwd: POINTER TO STRING;
	len:DINT;
END_VAR
VAR
	hFile: RTS_IEC_HANDLE;
	udiOpenError: RTS_IEC_RESULT;
	udiReadError: RTS_IEC_RESULT;
	udiWriteError: RTS_IEC_RESULT;
	i :INT;
	iTemp: UDINT;
	udiPos: UDINT;
	str_size: __XWORD;
	udiByteRead: UDINT;

	len_of_line: INT;
	len_of_number :INT;
	magicNumber:REAL;
	check_sum:REAL:= 0;
	temp_num:REAL;
	udiByteWrite: LWORD;
END_VAR


set_wifi_passwd := FALSE;

hFile := sysfileopen(szFile := '/userapp/wifi_passwd.txt', am := sysfile.AM_WRITE, pResult := ADR(udiOpenError));
IF hFile = RTS_INVALID_HANDLE THEN //创建文件失败
	RETURN;
END_IF

udiPos := SysFileSetPos(hFile:=hFile, ulOffset:=0);	
udiByteWrite := sysfile.SysFileWrite(hFile := hFile,pbyBuffer := passwd,ulSize := len, pResult := ADR(udiWriteError));
IF udiByteWrite = 0 THEN
	sysfile.SysFileClose(hFile := hFile);
	RETURN;
END_IF

sysfile.SysFileClose(hFile := hFile);
set_wifi_passwd := TRUE;
RETURN;

END_FUNCTION

// Device/Application/Functions/read_ip
FUNCTION read_ip : BOOL
VAR_INPUT
	ip: POINTER TO STRING;
END_VAR

VAR
	hFile: RTS_IEC_HANDLE;
	udiOpenError: RTS_IEC_RESULT;
	udiReadError: RTS_IEC_RESULT;
	i :INT;
	iTemp: UDINT;
	udiPos: UDINT;
	str_size: __XWORD;
	udiByteRead: LWORD;

	len_of_line: INT;
	len_of_number :INT;
	magicNumber:REAL;
	check_sum:REAL:= 0;
	temp_num:REAL;
END_VAR

read_ip := FALSE;

//检测文件是否存在
hFile := sysfileopen(szFile := '/userapp/ipaddr.txt', am := sysfile.AM_READ, pResult:= ADR(udiOpenError));
IF hFile = RTS_INVALID_HANDLE	THEN  //文件不存在
	RETURN;
END_IF
//文件存在，开始读取内容
udiPos := SysFileSetPos(hFile:=hFile, ulOffset := 0);
udiByteRead := sysfile.SysFileRead(hfile := hFile,pbyBuffer := ip, ulSize := 32, pResult := ADR(udiReadError));
IF udiByteRead < 4 THEN  //读取失败
	sysfile.SysFileClose(hFile := hFile);
	RETURN;
END_IF
sysfile.SysFileClose(hFile := hFile);
read_ip := TRUE;

END_FUNCTION

// Device/Application/Functions/read_wifi_passwd
FUNCTION read_wifi_passwd : BOOL
VAR_INPUT
	passwd: POINTER TO STRING;
END_VAR

VAR
	hFile: RTS_IEC_HANDLE;
	udiOpenError: RTS_IEC_RESULT;
	udiReadError: RTS_IEC_RESULT;
	i :INT;
	iTemp: UDINT;
	udiPos: UDINT;
	str_size: __XWORD;
	udiByteRead: LWORD;

	len_of_line: INT;
	len_of_number :INT;
	magicNumber:REAL;
	check_sum:REAL:= 0;
	temp_num:REAL;
END_VAR

read_wifi_passwd := FALSE;

//检测文件是否存在
hFile := sysfileopen(szFile := '/userapp/wifi_passwd.txt', am := sysfile.AM_READ, pResult:= ADR(udiOpenError));
IF hFile = RTS_INVALID_HANDLE	THEN  //文件不存在
	RETURN;
END_IF
//文件存在，开始读取内容
udiPos := SysFileSetPos(hFile:=hFile, ulOffset := 0);
udiByteRead := sysfile.SysFileRead(hfile := hFile,pbyBuffer := passwd, ulSize := 32, pResult := ADR(udiReadError));
IF udiByteRead < 4 THEN  //读取失败
	sysfile.SysFileClose(hFile := hFile);
	RETURN;
END_IF
sysfile.SysFileClose(hFile := hFile);
read_wifi_passwd := TRUE;

END_FUNCTION
